// TIA Portal V21 export
VAR_GLOBAL   // PLC tag table "K_Paratie"
END_VAR
VAR_GLOBAL CONSTANT   // user constants
   K_NumLinci : Int := 4;
END_VAR
